TEXTLIST TL_HeaderMachineState
  0 = 'Uninitialized'
  10 = 'Initializing'
  20 = 'Ready-Initialized'
  30 = 'Auto'
  40 = 'Auto to Manual'
  50 = 'Manual'
  60 = 'Manual to Auto'
  70 = 'Reset'
  80 = 'Reset done'
  -10 = 'Aborting'
  -20 = 'Emergency'
   = ''
END_TEXTLIST

(* stored: Version 1.1.0.1, ProductVersion 3.1.4024.9
   TextList TL_HeaderMachineState: Id {20719721-8fab-47e1-9421-902f9386afb1} *)
